INTERFACE ITF_ControlElement3 EXTENDS ITF_BaseControlElement

END_INTERFACE

(* stored: Version 1.1.0.1, ProductVersion 3.1.4024.15
   Itf ITF_ControlElement3: Id {6d23e08c-e94e-489b-a8c6-c9a5377ef5ed} *)
